// TIA Portal V19 export
TYPE "LAF_typeMachineInformation"
TITLE = typeUnitInformation
// Information about the unit
// stored: Access Published
   STRUCT
      equipmentID : DInt;   // Unique ID for all equipment in the plant / plant specific equipment identifier (defined by the project owner, ID can be written at commissioning
      equipmentName : WString;   // Equipment name by the Equipment Vendor
      equipmentVersion : WString;   // Vendor specific version of the equipment: syntax Vxx.xx.xxx
      interfaceVersionProject : WString;   // Project specific version of the interface: syntax Vxx.xx.xxx
      lineID : DInt;   // Line ID for all equipment in the Plant - project/ plant specific line identifier (defined by the Project owner, ID can be written at commissioning)
      vendorID : DInt;   // Unique vendor-supplier identifier of the equipment vendor
   END_STRUCT;
END_TYPE
